	8://Symbol exist and Value has changed
		byCounterWaitInStep_ReadAds := byCounterWaitInStep_ReadAds + 1;
			byCounterWaitInStep_ReadAds := LIMIT(1,byCounterWaitInStep_ReadAds,2);
	
		IF byCounterWaitInStep_ReadAds = 1 THEN 
			FOR udiLPCheckReadArrays_ReadAds := 1 TO udiNumberLoopHalf_ReadAds BY 1 DO
				IF stADSRead_ReadAds[udiLPCheckReadArrays_ReadAds].sFullSymbolName = stADSReadNew_ReadAds[udiLPCheckReadArrays_ReadAds].sFullSymbolName THEN
					stADSReadNew_ReadAds[udiLPCheckReadArrays_ReadAds].arrValue := stADSRead_ReadAds[udiLPCheckReadArrays_ReadAds].arrValue;
				END_IF
			END_FOR
		END_IF	
			IF byCounterWaitInStep_ReadAds = 2 AND udiNumberLoopFull_ReadAds <> udiNumberLoopHalf_ReadAds THEN 
				FOR udiLPCheckReadArrays_ReadAds := (udiNumberLoopHalf_ReadAds + 1) TO udiNumberLoopFull_ReadAds BY 1 DO
					IF stADSRead_ReadAds[udiLPCheckReadArrays_ReadAds].sFullSymbolName = stADSReadNew_ReadAds[udiLPCheckReadArrays_ReadAds].sFullSymbolName THEN
						stADSReadNew_ReadAds[udiLPCheckReadArrays_ReadAds].arrValue := stADSRead_ReadAds[udiLPCheckReadArrays_ReadAds].arrValue;	
					END_IF
				END_FOR
			END_IF 
		
				IF byCounterWaitInStep_ReadAds >= 2 THEN iState_ReadAds := 10; END_IF			
		
			//Timeout
			IF timTimout_ReadAds.Q THEN iState_ReadAds := 200; END_IF
		
	9://Copy the new symbol in the array
		byCounterWaitInStep_ReadAds := 0;
			stADSReadNew_ReadAds := stADSRead_ReadAds;
				iState_ReadAds := 10;
			
	10://Write in Buffer if the send bus is busy or send a messege if the buffer is not empty
		byCounterWaitInStep_ReadAds := 0;
	
		IF NOT Lynus_Standards.GVL_Communicator.arrInterfaceInfoValueSendTo[byReadWriteArrayNumber].bBusy THEN	
			Lynus_Standards.GVL_Communicator.arrInterfaceInfoValueSendTo[byReadWriteArrayNumber].arrValue := arrValueDefault_ReadAds; 						//Clear send Interface if it is no message to send
				Lynus_Standards.GVL_Communicator.arrInterfaceInfoValueSendTo[byReadWriteArrayNumber].sSymbolUnit := ''; 
					Lynus_Standards.GVL_Communicator.arrInterfaceInfoValueSendTo[byReadWriteArrayNumber].sFullSymbolName := '';
						Lynus_Standards.GVL_Communicator.arrInterfaceInfoValueSendTo[byReadWriteArrayNumber].sSymbolType := '';
							IF fbBuffer_ReadAds.nCount > 0 THEN							
								iState_ReadAds := 11;														//Send a new messege from the buffer
							END_IF																			
		END_IF
			IF ((Lynus_Standards.GVL_Communicator.arrInterfaceInfoValueSendTo[byReadWriteArrayNumber].bBusy OR fbBuffer_ReadAds.nCount = 0) AND NOT bValueIsTheSame_ReadAds) THEN
				iState_ReadAds := 20;																		//Insert a new value in the buffer if the send bus is busy or no value is stored in the buffer
			ELSE
				IF iState_ReadAds = 10 THEN 																						
					iState_ReadAds := 100;																	//Value is the same
				END_IF																						
			END_IF
		
			//Timeout
			IF timTimout_ReadAds.Q THEN iState_ReadAds := 200; END_IF
	
	11://Read out a Value from the buffer for sending
		IF udiCounterReadBuffer_New_ReadAds <> fbBuffer_ReadAds.nCount AND fbBuffer_ReadAds.bOk THEN
			udiCounterReadBuffer_New_ReadAds := fbBuffer_ReadAds.nCount;
				IF fbBuffer_ReadAds.cbReturn <= 2000 THEN 
					FOR udiLPCheckReadBuffer_ReadAds := 1 TO fbBuffer_ReadAds.cbReturn BY 1 DO	
						IF byCounterValueReadOut_ReadAds = 0 AND arrBufferRead_ReadAds[udiLPCheckReadBuffer_ReadAds] <> 59 THEN sSymbolNameOutFromBuffer_ReadAds := CONCAT(sSymbolNameOutFromBuffer_ReadAds,F_ToCHR(arrBufferRead_ReadAds[udiLPCheckReadBuffer_ReadAds])); END_IF 
							IF arrBufferRead_ReadAds[udiLPCheckReadBuffer_ReadAds] = 59 THEN byCounterValueReadOut_ReadAds := byCounterValueReadOut_ReadAds + 1; END_IF
								byCounterValueReadOut_ReadAds := LIMIT(0,byCounterValueReadOut_ReadAds,Lynus_Standards.Constants_Communicator.bySizeOfValueArray);
									IF byCounterValueReadOut_ReadAds >= 1 AND arrBufferRead_ReadAds[udiLPCheckReadBuffer_ReadAds] <> 59 AND arrBufferRead_ReadAds[udiLPCheckReadBuffer_ReadAds] <> 0 THEN 
										arrValueOutFromBuffer_ReadAds[byCounterValueReadOut_ReadAds] := CONCAT(arrValueOutFromBuffer_ReadAds[byCounterValueReadOut_ReadAds],F_ToCHR(arrBufferRead_ReadAds[udiLPCheckReadBuffer_ReadAds])); 
									END_IF    	
					END_FOR				 
						IF arrBufferRead_ReadAds[udiLPCheckReadBuffer_ReadAds] = 0 THEN iState_ReadAds := 12; byCounterValueReadOut_ReadAds := 0; END_IF
				END_IF
		END_IF
		
			IF timTimout_ReadAds.Q THEN iState_ReadAds := 200; END_IF
	
	12://Write the Date on interface and start the sending
		byCounterWaitInStep_ReadAds := byCounterWaitInStep_ReadAds + 1;
			byCounterWaitInStep_ReadAds := LIMIT(1,byCounterWaitInStep_ReadAds,2);
	
		IF byCounterWaitInStep_ReadAds = 1 THEN 
			FOR udiLPCheckVarInfoBeforSending_ReadAds := 1 TO udiNumberLoopHalf_ReadAds BY 1 DO
				IF Lynus_Standards.GVL_Communicator.arrInterfaceInfoAlVariables[byReadWriteArrayNumber,udiLPCheckVarInfoBeforSending_ReadAds].sFullSymbolName = sSymbolNameOutFromBuffer_ReadAds THEN
					Lynus_Standards.GVL_Communicator.arrInterfaceInfoValueSendTo[byReadWriteArrayNumber].sFullSymbolName := sSymbolNameOutFromBuffer_ReadAds;
						Lynus_Standards.GVL_Communicator.arrInterfaceInfoValueSendTo[byReadWriteArrayNumber].sSymbolUnit := Lynus_Standards.GVL_Communicator.arrInterfaceInfoAlVariables[byReadWriteArrayNumber,udiLPCheckVarInfoBeforSending_ReadAds].sSymbolUnit;
							Lynus_Standards.GVL_Communicator.arrInterfaceInfoValueSendTo[byReadWriteArrayNumber].sSymbolType := Lynus_Standards.GVL_Communicator.arrInterfaceInfoAlVariables[byReadWriteArrayNumber,udiLPCheckVarInfoBeforSending_ReadAds].sSymbolType;
								Lynus_Standards.GVL_Communicator.arrInterfaceInfoValueSendTo[byReadWriteArrayNumber].arrValue := arrValueOutFromBuffer_ReadAds;
									Lynus_Standards.GVL_Communicator.arrInterfaceInfoValueSendTo[byReadWriteArrayNumber].bBusy := TRUE;
										iState_ReadAds := 13;
											EXIT;	
				END_IF 		 	   	
			END_FOR 	
		END_IF
			IF byCounterWaitInStep_ReadAds = 2 AND udiNumberLoopFull_ReadAds <> udiNumberLoopHalf_ReadAds THEN 
				FOR udiLPCheckVarInfoBeforSending_ReadAds := (udiNumberLoopHalf_ReadAds + 1) TO udiNumberLoopFull_ReadAds BY 1 DO
					IF Lynus_Standards.GVL_Communicator.arrInterfaceInfoAlVariables[byReadWriteArrayNumber,udiLPCheckVarInfoBeforSending_ReadAds].sFullSymbolName = sSymbolNameOutFromBuffer_ReadAds THEN
						Lynus_Standards.GVL_Communicator.arrInterfaceInfoValueSendTo[byReadWriteArrayNumber].sFullSymbolName := sSymbolNameOutFromBuffer_ReadAds;
							Lynus_Standards.GVL_Communicator.arrInterfaceInfoValueSendTo[byReadWriteArrayNumber].sSymbolUnit := Lynus_Standards.GVL_Communicator.arrInterfaceInfoAlVariables[byReadWriteArrayNumber,udiLPCheckVarInfoBeforSending_ReadAds].sSymbolUnit;
								Lynus_Standards.GVL_Communicator.arrInterfaceInfoValueSendTo[byReadWriteArrayNumber].sSymbolType := Lynus_Standards.GVL_Communicator.arrInterfaceInfoAlVariables[byReadWriteArrayNumber,udiLPCheckVarInfoBeforSending_ReadAds].sSymbolType;
									Lynus_Standards.GVL_Communicator.arrInterfaceInfoValueSendTo[byReadWriteArrayNumber].arrValue := arrValueOutFromBuffer_ReadAds;
										Lynus_Standards.GVL_Communicator.arrInterfaceInfoValueSendTo[byReadWriteArrayNumber].bBusy := TRUE;
											iState_ReadAds := 13;
												EXIT;	
					END_IF 		 	   	
				END_FOR 	
			END_IF
		
			IF timTimout_ReadAds.Q THEN iState_ReadAds := 200; END_IF
			
	13://Clear Read Buffer (conserve resources because the code must also work for small plc's)
		byCounterWaitInStep_ReadAds := 0;
			sSymbolNameOutFromBuffer_ReadAds := '';
				MEMCPY(ADR(arrBufferRead_ReadAds),ADR(arrBufferWriteReadDefault_ReadAds),SIZEOF(arrBufferRead_ReadAds));
					arrValueOutFromBuffer_ReadAds := arrValueDefault_ReadAds;
		
			iState_ReadAds := 10;
			
	20://Dim size from the values and symbol name befor can saving in buffer
		uiNumberValueSymbolSize_ReadAds := 0;
			byNumberOfValues_ReadAds_ReadAds := 0;
				byLenghSymbolName_ReadAds := 0;
		FOR byLPDimValueNumberASize_ReadAds := 1 TO Lynus_Standards.Constants_Communicator.bySizeOfValueArray BY 1 DO
			uiNumberValueSymbolSize_ReadAds := uiNumberValueSymbolSize_ReadAds + INT_TO_UINT(LEN(stADSReadNew_ReadAds[udiActiveNumberOfSymbol_ReadAds].arrValue[byLPDimValueNumberASize_ReadAds]));
				IF stADSReadNew_ReadAds[udiActiveNumberOfSymbol_ReadAds].arrValue[byLPDimValueNumberASize_ReadAds] <> '' THEN uiNumberValueSymbolSize_ReadAds := uiNumberValueSymbolSize_ReadAds + 1; END_IF 	
					IF stADSReadNew_ReadAds[udiActiveNumberOfSymbol_ReadAds].arrValue[byLPDimValueNumberASize_ReadAds] <> '' THEN byNumberOfValues_ReadAds_ReadAds := byNumberOfValues_ReadAds_ReadAds + 1; END_IF	
		END_FOR 	
			byLenghSymbolName_ReadAds := INT_TO_BYTE(LEN(stADSReadNew_ReadAds[udiActiveNumberOfSymbol_ReadAds].sFullSymbolName));
				uiNumberValueSymbolSize_ReadAds := uiNumberValueSymbolSize_ReadAds + byLenghSymbolName_ReadAds + 1;
		
			IF byNumberOfValues_ReadAds_ReadAds <= Lynus_Standards.Constants_Communicator.bySizeOfValueArray THEN
				FOR byLPDimLenghValues_ReadAds := 1 TO byNumberOfValues_ReadAds_ReadAds BY 1 DO
					arrLenghEachValue_ReadAds[byLPDimLenghValues_ReadAds] := INT_TO_BYTE(LEN(stADSReadNew_ReadAds[udiActiveNumberOfSymbol_ReadAds].arrValue[byLPDimLenghValues_ReadAds]));	
				END_FOR 
			END_IF
	
		IF byNumberOfValues_ReadAds_ReadAds <= Lynus_Standards.Constants_Communicator.bySizeOfValueArray AND byNumberOfValues_ReadAds_ReadAds >= 1 AND uiNumberValueSymbolSize_ReadAds <> 0 THEN iState_ReadAds := 21; END_IF
		
			IF timTimout_ReadAds.Q THEN iState_ReadAds := 200; END_IF
			
	21://String to Ascii Symbol Name and values
		IF byLenghSymbolName_ReadAds <= 49 THEN
			FOR byLPSymbolNameToAscii_ReadAds := 1 TO byLenghSymbolName_ReadAds BY 1 DO
				arrSymbolName_ReadAds[byLPSymbolNameToAscii_ReadAds] := F_ToASC(MID(stADSReadNew_ReadAds[udiActiveNumberOfSymbol_ReadAds].sFullSymbolName,1,byLPSymbolNameToAscii_ReadAds));
			END_FOR 
		END_IF
			IF byLenghSymbolName_ReadAds < 49 THEN arrSymbolName_ReadAds[byLenghSymbolName_ReadAds + 1] := F_ToASC(';'); END_IF  	
		
		IF byNumberOfValues_ReadAds_ReadAds <= Lynus_Standards.Constants_Communicator.bySizeOfValueArray THEN 
			FOR byLPValueNameToAscii_1_ReadAds := 1 TO byNumberOfValues_ReadAds_ReadAds BY 1 DO
				IF arrLenghEachValue_ReadAds[byLPValueNameToAscii_1_ReadAds] <= 31 THEN 
					FOR byLPValueNameToAscii_2_ReadAds := 1 TO arrLenghEachValue_ReadAds[byLPValueNameToAscii_1_ReadAds] BY 1 DO
						arrValueName_ReadAds[byLPValueNameToAscii_1_ReadAds,byLPValueNameToAscii_2_ReadAds] := F_ToASC(MID(stADSReadNew_ReadAds[udiActiveNumberOfSymbol_ReadAds].arrValue[byLPValueNameToAscii_1_ReadAds],1,byLPValueNameToAscii_2_ReadAds));
					END_FOR
				END_IF
					arrValueName_ReadAds[byLPValueNameToAscii_1_ReadAds,byLPValueNameToAscii_2_ReadAds] := F_ToASC(';'); 			
			END_FOR 
		END_IF 
		
		IF byLenghSymbolName_ReadAds <= 49 AND byNumberOfValues_ReadAds_ReadAds <= Lynus_Standards.Constants_Communicator.bySizeOfValueArray AND arrLenghEachValue_ReadAds[byNumberOfValues_ReadAds_ReadAds] <= 31 THEN iState_ReadAds := 22; END_IF
		
			IF timTimout_ReadAds.Q THEN iState_ReadAds := 200; END_IF	
			
	22://Prepare Write array for Buffer
		IF byLenghSymbolName_ReadAds <= 48 THEN
			FOR uiLPWriteByteValueInArray_ReadAds := 1 TO (byLenghSymbolName_ReadAds + 1) BY 1 DO
				arrBufferWrite_ReadAds[uiLPWriteByteValueInArray_ReadAds] := arrSymbolName_ReadAds[uiLPWriteByteValueInArray_ReadAds];
			END_FOR 
		END_IF
		
		IF byLenghSymbolName_ReadAds <= 48 THEN	iState_ReadAds := 23; END_IF
			
			IF timTimout_ReadAds.Q THEN iState_ReadAds := 200; END_IF
	
	23://Prepare Write array for Buffer
		uiValueForLoopStart_ReadAds := uiLPWriteByteValueInArray_ReadAds;
			byValueInTurn_ReadAds := byValueInTurn_ReadAds + 1;
				byValueInTurn_ReadAds := LIMIT(1,byValueInTurn_ReadAds,Lynus_Standards.Constants_Communicator.bySizeOfValueArray);
					uiValueForLoopStop_ReadAds := arrLenghEachValue_ReadAds[byValueInTurn_ReadAds] + uiValueForLoopStart_ReadAds;
						byCounterValue_ReadAds := 0;
							
							IF uiValueForLoopStart_ReadAds >= 1 AND uiValueForLoopStart_ReadAds <= 2000 AND uiValueForLoopStop_ReadAds >= 1 AND uiValueForLoopStop_ReadAds <= 2000 THEN 
								FOR uiLPWriteByteValueInArray_ReadAds := uiValueForLoopStart_ReadAds TO uiValueForLoopStop_ReadAds BY 1 DO
									byCounterValue_ReadAds :=  byCounterValue_ReadAds + 1;
										byCounterValue_ReadAds := LIMIT(1,byCounterValue_ReadAds,31);	
											arrBufferWrite_ReadAds[uiLPWriteByteValueInArray_ReadAds] := arrValueName_ReadAds[byValueInTurn_ReadAds,byCounterValue_ReadAds];
								END_FOR 
							END_IF
		
		IF byValueInTurn_ReadAds >= byNumberOfValues_ReadAds_ReadAds AND uiValueForLoopStart_ReadAds >= 1 AND uiValueForLoopStart_ReadAds <= 2000 AND uiValueForLoopStop_ReadAds >= 1 AND uiValueForLoopStop_ReadAds <= 2000 THEN 
			iState_ReadAds := 24; 
				uiValueForLoopStart_ReadAds := 0;
					byValueInTurn_ReadAds := 0;
						uiValueForLoopStop_ReadAds := 0;
							byCounterValue_ReadAds := 0;			
		END_IF
			
			IF timTimout_ReadAds.Q THEN iState_ReadAds := 200; END_IF

	24://Write Value in Buffer
		iState_ReadAds := 25; 
				
	25://Check if the new value is stored in the buffer
		IF fbBuffer_ReadAds.bOk AND fbBuffer_ReadAds.nCount <> udiCounterReadBuffer_New_ReadAds THEN udiCounterReadBuffer_New_ReadAds := fbBuffer_ReadAds.nCount; iState_ReadAds := 26; END_IF  	
			
			IF timTimout_ReadAds.Q THEN iState_ReadAds := 200; END_IF
		
	26://Clear the Write Buffer (conserve resources because the code must also work for small plc's)
		MEMCPY(ADR(arrBufferWrite_ReadAds),ADR(arrBufferWriteReadDefault_ReadAds),SIZEOF(arrBufferWrite_ReadAds));
		
			iState_ReadAds := 100;

	100://Check for other variable
		//Next symbol
		IF udiActiveNumberOfSymbol_ReadAds < Lynus_Standards.GVL_Communicator.arrCounterVariableInArray[byReadWriteArrayNumber] AND udiNumberInProgress_ReadAds < udiNumberSizeValues_ReadAds THEN iState_ReadAds := -4; udiNumberInProgress_ReadAds := udiNumberInProgress_ReadAds + 1; END_IF
			//Start with the next 10 Variables
			IF (udiNumberInProgress_ReadAds >= udiNumberSizeValues_ReadAds AND iState_ReadAds = 100) THEN 
				iState_ReadAds := -8; 
					udiNumberInProgress_ReadAds := 0;
			END_IF	
				//Start from New with the first 10 Variables 	
				IF udiActiveNumberOfSymbol_ReadAds >= Lynus_Standards.GVL_Communicator.arrCounterVariableInArray[byReadWriteArrayNumber] THEN
					iState_ReadAds := -8; 
						udiActiveNumberOfSymbol_ReadAds := 0;
							udiNumberInProgress_ReadAds := 0;
								udiRestValueSymbolRead_ReadAds := 0;
						 			bFirstReadCycleDone_ReadAds := TRUE; 
				END_IF			
			
			bError_ReadAds := FALSE;
				uiInternError_ReadAds := 0;
			
			IF timTimout_ReadAds.Q THEN iState_ReadAds := 200; END_IF
				
	200://Error
		bError_ReadAds := TRUE; fbADSREADWRITE_ReadAds.WRTRD := FALSE; bValueIsTheSame_ReadAds := FALSE; 
			udiActiveNumberOfSymbol_ReadAds := 0; byCounterWaitInStep_ReadAds := 0; udiNumberInProgress_ReadAds := 0; udiRestValueSymbolRead_ReadAds := 0;
		
		//Clear the write Buffer befor go to step 0 (conserve resources because the code must also work for small plc's)
		MEMCPY(ADR(arrBufferWrite_ReadAds),ADR(arrBufferWriteReadDefault_ReadAds),SIZEOF(arrBufferWrite_ReadAds));
		
		//Clear the read Buffer befor go to step 0 (conserve resources because the code must also work for small plc's)
		sSymbolNameOutFromBuffer_ReadAds := '';
			MEMCPY(ADR(arrBufferRead_ReadAds),ADR(arrBufferWriteReadDefault_ReadAds),SIZEOF(arrBufferRead_ReadAds));
				arrValueOutFromBuffer_ReadAds := arrValueDefault_ReadAds;
			
		//Count up when an error has occurred
		byErrorCounter_ReadAds := byErrorCounter_ReadAds + 1;		
				
			iState_ReadAds := 300;
	
	300://Wait in Error and clear the rest from the read and write buffer (conserve resources because the code must also work for small plc's)
		byCounterWaitInStep_ReadAds := byCounterWaitInStep_ReadAds + 1;
	
			//Restart new from in Step -8. No Reset from the complete System
			IF byCounterWaitInStep_ReadAds > 10 AND byErrorCounter_ReadAds <= 10 THEN byCounterWaitInStep_ReadAds := 0; iState_ReadAds := -8; END_IF
				//Restart new from in Step -10. Reset from the complete System after to much Errors
				IF byCounterWaitInStep_ReadAds > 10 AND byErrorCounter_ReadAds > 10 THEN 
						byCounterWaitInStep_ReadAds := 0; 
							//Reset Read Steps and start from new
							iState_ReadAds := -10;
								//Reset Write Steps and start from new
								iState_WriteAds := -2;
									byErrorCounter_ReadAds := 0; 
				END_IF
	
END_CASE	

//Resetting the error counter after not being in the error step for 30 min
timResetErrorCounter_ReadAds(IN:= byErrorCounter_ReadAds <> 0, PT:= T#30M, Q=> , ET=> );
	IF timResetErrorCounter_ReadAds.Q THEN byErrorCounter_ReadAds := 0; END_IF 

//Read Out Variable by ADS
fbADSREADWRITE_ReadAds(
	NETID:= fbNedID.AddrString, 
	PORT:= uiPort, 
	IDXGRP:= 16#F080, 
	IDXOFFS:= udiNumberSizeValues_ReadAds, 
	WRITELEN:= , 
	READLEN:= udiSizeReq_ReadAds, 
	SRCADDR:= , 
	DESTADDR:= ADR(arrValueRead_ReadAds), 
	WRTRD:= , 
	TMOUT:= T#5S, 
	BUSY=> , 
	ERR=> , 
	ERRID=> );

FPErrorReadWrite_ReadAds(CLK:= fbADSREADWRITE_ReadAds.ERR, Q=> );	
	
//Buffer Read Value from ADS
FPWriteValueToBufferStep25_ReadAds(CLK:= iState_ReadAds = 24, Q=> );
FPReadValueToBufferStep11_ReadAds(CLK:= iState_ReadAds = 11, Q=> );

IF FPReadValueToBufferStep11_ReadAds.Q THEN fbBuffer_ReadAds.A_RemoveHead(); END_IF
IF FPWriteValueToBufferStep25_ReadAds.Q THEN fbBuffer_ReadAds.A_AddTail(); END_IF

//Reset the Buffer after a Buffer Overflow
IF fbBuffer_ReadAds.nCount <> 0 AND NOT fbBuffer_ReadAds.bOk THEN timResetBuffer_ReadAds.IN := TRUE; ELSE timResetBuffer_ReadAds.IN := FALSE; END_IF
	timResetBuffer_ReadAds(IN:= , PT:= T#40S, Q=> , ET=> );
		IF timResetBuffer_ReadAds.Q THEN fbBuffer_ReadAds.A_Reset(); END_IF

fbBuffer_ReadAds(
	pWrite:= ADR(arrBufferWrite_ReadAds), 
	cbWrite:= uiNumberValueSymbolSize_ReadAds, 
	pRead:= ADR(arrBufferRead_ReadAds), 
	cbRead:= SIZEOF(arrBufferRead_ReadAds), 
	pBuffer:= ADR(arrBufferADSRead_ReadAds), 
	cbBuffer:= SIZEOF(arrBufferADSRead_ReadAds), 
	bOk=> Lynus_Standards.GVL_Communicator.arrInterfaceInfoValueSendTo[byReadWriteArrayNumber].bBufferOK, 
	nCount=> Lynus_Standards.GVL_Communicator.arrInterfaceInfoValueSendTo[byReadWriteArrayNumber].udiCountBuffer, 
	cbSize=> , 
	cbReturn=> );

END_IF
	
//Busy
IF iState_ReadAds >= -8 OR iState_WriteAds >= 0 THEN bBusy := TRUE; ELSE bBusy := FALSE; END_IF
	
//Error
IF (bError_ReadAds AND iState_ReadAds <> - 10 AND iState_ReadAds <> - 9) OR (bError_WriteAds AND iState_WriteAds <> - 1 AND iState_WriteAds <> - 2) THEN fbErrorCodes.bErrorIntern := TRUE; ELSE fbErrorCodes.bErrorIntern := FALSE; END_IF

IF fbADSREADWRITE_ReadAds.ERR OR fbADSREADWRITE_WriteAds.ERR OR fbADSWrite_WriteAds.ERR THEN fbErrorCodes.bErrorADS := TRUE; END_IF

IF fbADSREADWRITE_ReadAds.ERR THEN fbErrorCodes.udiErrorCodeADS := fbADSREADWRITE_ReadAds.ERRID; END_IF
IF fbADSREADWRITE_WriteAds.ERR THEN fbErrorCodes.udiErrorCodeADS := fbADSREADWRITE_WriteAds.ERRID; END_IF
IF fbADSWrite_WriteAds.ERR THEN fbErrorCodes.udiErrorCodeADS := fbADSWrite_WriteAds.ERRID; END_IF

IF NOT fbADSREADWRITE_ReadAds.ERR AND NOT fbADSREADWRITE_ReadAds.BUSY AND NOT
	fbADSREADWRITE_WriteAds.ERR AND NOT fbADSREADWRITE_WriteAds.BUSY AND NOT fbADSWrite_WriteAds.ERR AND NOT fbADSWrite_WriteAds.BUSY THEN 
		fbErrorCodes.bErrorADS := FALSE;
			fbErrorCodes.udiErrorCodeADS := 0; 
END_IF 	     
	
fbErrorCodes(
	bErrorADS:= , 
	bErrorIntern:= , 
	udiErrorCodeADS:= , 
	udiErrorCodesInternRead:= uiInternError_ReadAds, 
	udiErrorCodesInternWrite:= uiInternError_WriteAds, 
	udiErrorCodeADS_Out=> udiErrorCodeOut, 
	bError=> bError, 
	eErrorReadWrite_Out=> eErrorReadWrite_Out);
	
// interval sending
// define what is selected
CASE eUploadType OF
	0: 	m_EnableChange_upload	:= FALSE;
		m_EnableInterval		:= TRUE;
		time_Interval			:= T#5M;
	1: 	m_EnableChange_upload	:= FALSE;
		m_EnableInterval		:= TRUE;
		time_Interval			:= T#1M;	
	2: 	m_EnableChange_upload	:= TRUE;
		m_EnableInterval		:= FALSE;
		time_Interval			:= T#5M;
	3: 	m_EnableChange_upload	:= TRUE;
		m_EnableInterval		:= TRUE;
		time_Interval			:= T#5M;	
	4: 	m_EnableChange_upload	:= TRUE;
		m_EnableInterval		:= TRUE;
		time_Interval			:= T#1M;	
END_CASE

// m_TriggerIntervalSend and m_EnableChange_upload used in line 997/996, 1011/1010 & 1606/1605

timer_Interval(IN:=NOT m_TriggerIntervalSend AND m_EnableInterval, PT:=time_Interval);
		
IF udiActiveNumberOfSymbol_ReadAds=udiNumberLoopFull_ReadAds AND iState_ReadAds>12 AND m_TriggerIntervalSend=TRUE  AND bFirstReadCycleDone_ReadAds THEN
	m_TriggerIntervalSend:=FALSE;
END_IF
IF (timer_interval.Q AND udiActiveNumberOfSymbol_ReadAds =0) THEN
	m_TriggerIntervalSend:=TRUE;
END_IF

END_FUNCTION_BLOCK

(* stored: Version 1.1.0.1, ProductVersion 3.1.4024.11
   POU FB_ReadWrite_V2: Id {2050f89d-b715-4b84-a913-a7f6d6b09577}, SpecialFunc None *)
